// TIA Portal V20 export
// export: Created 2025-12-01T14:57:22.4882331Z, ExportSetting None, DisplayName Totally Integrated Automation Portal, DisplayVersion V20 Update 3, DisplayName TIA Portal Openness, DisplayVersion V20 Update 3, DisplayName TIA Portal Version Control Interface, DisplayVersion V20 Update 3, DisplayName STEP 7 Professional, DisplayVersion V20 Update 3, DisplayName STEP 7 Safety, DisplayVersion V20 Update 2, DisplayName WinCC Basic/Comfort/Advanced, DisplayVersion V20 Update 3, DisplayName WinCC Professional, DisplayVersion V20 Update 3, DisplayName WinCC Unified, DisplayVersion V20 Update 3
FUNCTION "FC970_Datos_Sinoptico" : Void   // FC970, LAD
TITLE = Datos Generales para la Pantalla
{ S7_Optimized_Access := 'FALSE' }
AUTHOR : PANTALLA
NAME : 20180615
VERSION : 4.3
// =- Inicializar Variables
// - Transferencia del Estado del VI para la Pantallaf
// - Nieves modificado para minimizar lineas de código
// - inicialización de Variables de mesa
// stored: AutoNumber false, SetENOAutomatically false
   VAR_INPUT
      NumDB_Sinoptico : UInt;   // DB de envio estado zonas y mesas a Pantalla
      Offset_InfoMesas : UInt;   // Byte Inicio zona de Informacion de Mesas a Pantalla
      Offset_NumUTsMesas : UInt;   // Byte Inicio zona de Numero de UTs en Mesa para Pantalla
   END_VAR
   VAR_TEMP
      ByteMesa : Struct
         Vacia : Bool;
         Cargada : Bool;
         En_Descarga : Bool;
         En_Carga : Bool;
         Etapas_Reset : Bool;
         Paro : Bool;
         Manual : Bool;
         En_Error : Bool;
      END_STRUCT;
      P_ByteMesa : DWord;
      P_Temporal : DWord;
      CNT_NumMesa : UInt;
      DB_Sinoptico : Word;
      NumeroUTs : UInt;
      NumeroUT : UInt;
      Tmp_Estado_Mesa : "EstadosMesa";
      Tmp_Estado_Maquina : "EstadoMaquina";
   END_VAR
BEGIN

NETWORK
TITLE = Inicializar Variables
// ------------------------------------------------------------------------
// --- Inicializar Variabes

      L     #NumDB_Sinoptico;  // DB Estado Zona
      T     #DB_Sinoptico;

      L     0;  // Iniciamos el contador de Mesas
      T     #CNT_NumMesa;


NETWORK
TITLE = Transferencia del Estado del VI para la Pantalla
// ------------------------------------------------------------------------
// --- Recogo el estado del VI (Mesa

BFIF: NOP   0;
// ------------------------------------------------------------------
// ---- Recoger las variables que se necesitan

      L     P##ByteMesa;  // Inicializar
      T     #P_ByteMesa;
      L     0;
      T     LB [#P_ByteMesa];

// pasamos a evaluar el estado de la mesa
// ---- 1º - Si Esta en Error
      SET;
      A     "DB900_Estado_Mesas".EstadoVI[#CNT_NumMesa].Error_Mx;
      O     "DB904_Estado_Maquinas".EstadoVI[#CNT_NumMesa].Error_MAQx;
      =     #ByteMesa.En_Error;  // Mesa En Error

// --- Si la mesa está en modo mantenimiento. NIEVES MANTENIMIENTO
      SET;
      A     "DB902_Estado_ZonaMesa".EstadoMesas[#CNT_NumMesa].Mantenimiento_CBx;
      =     #ByteMesa.Manual;
      =     #ByteMesa.Paro;
      JC    nxt;

// FIN NIEVES MANTENIMIENTO

// ---- 3º - Si Esta en Manual
      SET;
      A     "DB900_Estado_Mesas".EstadoVI[#CNT_NumMesa].Manual;
      =     #ByteMesa.Manual;
      JC    nxt;  // si está en manual no puede estar en paro

// ---- 4º - Si Esta en Paro
      SET;
      A     "DB902_Estado_ZonaMesa".EstadoMesas[#CNT_NumMesa].Paro_CBx;
      AN    #ByteMesa.Manual;  // Mesa no esta en Manual
      =     #ByteMesa.Paro;


// ---- 2º - Si Esta en Reset
// NIEVES, CAMBIO EL ORDEN PORQUE SI ESTÁ EN RESET NO ES NECESARIO SEGUIR EVALUANDO MÁS CONDICIONES

nxt:  SET;
      A     "DB900_Estado_Mesas".EstadoVI[#CNT_NumMesa].Etapas_Reset;
      =     #ByteMesa.Etapas_Reset;  // Mesa Reset
      JC    nxt2;  // salta directamente a guardar el estado en el db
// ---- 5º - Si Esta en Vacia

      SET;
      A     "DB900_Estado_Mesas".EstadoVI[#CNT_NumMesa].Etapa_Vacia;
      =     #ByteMesa.Vacia;  // Mesa Vacia
      JC    nxt2;  // si está vacía no puede estar ni cargada ni en carga ni en descarga

// ---- 6º - Si Esta en Cargada
      SET;
      A     "DB900_Estado_Mesas".EstadoVI[#CNT_NumMesa].Etapa_Cargada;
      =     #ByteMesa.Cargada;  // Mesa Cargada, no puede estar ni en carga ni en descarga
      JC    nxt2;

// ---- 7º - Si Esta en Descarga
      SET;
      A     "DB900_Estado_Mesas".EstadoVI[#CNT_NumMesa].Etapas_Descarga_S0;
      O     "DB900_Estado_Mesas".EstadoVI[#CNT_NumMesa].Etapas_Descarga_S1;
      O     "DB900_Estado_Mesas".EstadoVI[#CNT_NumMesa].Etapas_Descarga_S2;
      O     "DB900_Estado_Mesas".EstadoVI[#CNT_NumMesa].Etapas_Descarga_S3;
      O     "DB900_Estado_Mesas".EstadoVI[#CNT_NumMesa].Etapas_Descarga_S4;
      =     #ByteMesa.En_Descarga;  // Mesa En Descarga evaluamos la carga por si está en simultaneo
      JC    nxt2;

// ---- 8º - Si Esta en Carga
      SET;
      A     "DB900_Estado_Mesas".EstadoVI[#CNT_NumMesa].Etapas_Carga_E0;
      O     "DB900_Estado_Mesas".EstadoVI[#CNT_NumMesa].Etapas_Carga_E1;
      O     "DB900_Estado_Mesas".EstadoVI[#CNT_NumMesa].Etapas_Carga_E2;
      O     "DB900_Estado_Mesas".EstadoVI[#CNT_NumMesa].Etapas_Carga_E3;
      O     "DB900_Estado_Mesas".EstadoVI[#CNT_NumMesa].Etapas_Carga_E4;
      =     #ByteMesa.En_Carga;  // Mesa En Carga
      JC    nxt2;

// ------------------------------------------------------------------------
// --- Cargo el Estado del VI (Mesa) en DB Sinoptico

nxt2: L     #CNT_NumMesa;  // Puntero Origen de Datos
      L     #Offset_InfoMesas;
      +D;
      SLD   3;
      T     #P_Temporal;

      OPN   DB [#DB_Sinoptico];  // Abrir DB Destino
      L     LB [#P_ByteMesa];  // Pasarselo
      T     DBB [#P_Temporal];



NETWORK
TITLE = Calculo y Transferencia del numero de UTs en una mesa para la Pantalla
// ------------------------------------------------------------------------
// --- Calculo de la cantidad de UT's por mesa
// ----------------------------------------------------------------------------

      CALL  "FC871_NumUTsEnMesa"
      ( Mesa   := #CNT_NumMesa,
        NumUTs := #NumeroUTs
      );

// ------------------------------------------------------------------------
// --- Cargo el numero de UT's en el DB Sinoptico

      L     #CNT_NumMesa;  // Puntero Origen de Datos
      L     #Offset_NumUTsMesas;
      +D;
      SLD   3;
      T     #P_Temporal;

      OPN   DB [#DB_Sinoptico];  // Abrir DB Destino

      L     #NumeroUTs;  // Pasarselo
      T     DBB [#P_Temporal];



NETWORK
TITLE = pasar a la siguiente mesa
// ------------------------------------------------------------------------
// ------------------------------------------------------------------------
// ------------------------------------------------------------------------
// --- Pasar a la Siguiente Mesa

      L     #CNT_NumMesa;
      L     "CTE_MaxMesas";  // Si no quedan Mesas ?
      >=I;
      JC    _END;

      L     1;  //Incrementa el contador de posicion
      L     #CNT_NumMesa;
      +I;
      T     #CNT_NumMesa;

      JU    BFIF;

// ------------------------------------------------------------------------
// --- Final de la Funcion

_END: NOP   0;


END_FUNCTION
